Staubli VAL3: start.pgx

program start()
begin
  call exo11()
end
